// TIA Portal V17 export
// export: Created 2021-12-03T08:13:20.4490419Z, ExportSetting WithDefaults, DisplayName Totally Integrated Automation Portal, DisplayVersion V17, DisplayName TIA Portal Openness, DisplayVersion V17, DisplayName TIA Portal Version Control Interface, DisplayVersion V17, DisplayName STEP 7 Professional, DisplayVersion V17, DisplayName STEP 7 Safety, DisplayVersion V17, DisplayName WinCC Advanced, DisplayVersion V17
DATA_BLOCK "GDB_Default_Set"   // DB2000
VERSION : 0.1
// stored: AutoNumber false, IsOnlyStoredInLoadMemory false, IsWriteProtectedInAS false
   VAR
      AccChiller : Struct   // Значения для чиллера ускорителя
         ChilPwrOnTm_PT : Int := 5;   // Время подготовки чиллера м
         ChilPwrOffTm_PT : Int := 10;   // Время охлаждения чиллера м
      END_STRUCT;
      FrqConv : Struct   // Уставки для преобразователя
         FstSpd : Int := 400;   // Быстрая скорость
         LwSpd : Int := 200;   // Медленная скорость
         Ramp : Int := 100;   // Рампа
      END_STRUCT;
      ScanSeqSet : Struct   // Уставки для
         CycleTime : Int := 120;   // Время цикла
         RfOn : Int := 3;   // Время задержки в СВЧ
         XrayOn : Int := 5;   // Время задержки в торм. излучении
      END_STRUCT;
   END_VAR
BEGIN
END_DATA_BLOCK
